{attribute 'qualified_only'}
{attribute 'strict'}
TYPE E_MixitMode :
(
	Mode_Off 	:= 0,
	Mode_Auto	:= 1,
	Mode_Manual	:= 2
);
END_TYPE

(* stored: Version 1.1.0.1, ProductVersion 3.1.4024.15
   DUT E_MixitMode: Id {1a7c5d5e-1834-442d-9499-28db3bc1cfc4} *)
